{attribute addProperty BoxType "KL6211-0004"}
{attribute addProperty Id "Channel_1Channel_8A16238100"}
{attribute addProperty CRC "343679516"}
{attribute addProperty SizeInBites "0"}
{attribute addProperty SizeInBytes "0"}
TYPE KL_147C221C :
STRUCT
	{attribute addProperty Name "Channel_1"}
	Channel_1 : Channel_8A162381;
END_STRUCT
END_TYPE

(* stored: Version 1.2.0.0, ProductVersion 3.1.4024.9
   DUT KL_147C221C: Id {143d0f7a-50b0-414c-8c7c-24665bc59669} *)
